Yaskawa INFORM job: R1_W01(KAMERA)(0,-90).JBI

/JOB
//NAME R1_W01(KAMERA)(0,-90)
//POS
///NPOS 10,10,0,0,0,0
///TOOL 0
///POSTYPE PULSE
///PULSE
C00000=-3259,-159822,-135039,10688,361,77457
C00001=-3259,-159822,-135039,10688,361,77457
C00002=-118675,-45665,-102005,21757,75350,73909
C00003=-180273,41623,-63008,27819,115689,72022
C00004=-173474,31677,-49799,19899,113315,69231
C00005=-168661,44467,-36169,18018,110829,70097
C00006=-171137,33845,-43401,22454,103512,69827
C00007=-168805,46512,-36363,18230,111966,70243
C00008=-168950,50616,-36887,18653,114300,70595
C00009=-169262,14064,-103081,21827,78231,74428
BC00000=159764,444967,1049074
BC00001=159764,23329,1049074
BC00002=282627,8095,1066129
BC00003=347792,15,1075175
BC00004=341835,15,1075175
BC00005=341835,15,1075175
BC00006=341836,15,1075173
BC00007=342000,15,1075175
BC00008=341884,15,1075175
BC00009=381794,1295,1075175
//INST
///DATE 2024/11/28 10:02
///ATTR SC,RW
///GROUP1 RB1,BS1
NOP
'r1_W01(kamera)(0,-90)
'Path W401
SFTOF
MOVJ C00000 BC00000 VJ=100.00
MOVJ C00001 BC00001 VJ=100.00
MOVJ C00002 BC00002 VJ=100.00
MOVJ C00003 BC00003 VJ=70.00
MOVJ C00004 BC00004 VJ=20.00 PL=0
MACRO1 MJ#(0) ARGF6
ARCON
WVON WEV#(2)
MOVL C00005 BC00005 V=10.0
MOVL C00006 BC00006 V=10.0
ARCOF
WVOF
MOVL C00007 BC00007 V=100.0
MOVL C00008 BC00008 V=166.7
MOVJ C00009 BC00009 VJ=100.00
END
